FUNCTION_BLOCK FB_InRange
VAR_INPUT
	i_fValue : LREAL;
	i_fRange : LREAL;
END_VAR
VAR_OUTPUT
END_VAR
VAR
	nCntAuto : UINT;
	nCntManual : UINT;
	nCntMaintenance : UINT;
	
END_VAR


SUPER^.m_Main();

END_FUNCTION_BLOCK

(* stored: Version 1.1.0.1, ProductVersion 3.1.4024.12
   POU FB_InRange: Id {49259daf-98ab-4b7a-8dd3-2d45bf56c0dc}, SpecialFunc None *)
